	110:   
		   IF Ref_MachineStateModel.Sts_Stopping AND Ref_Unit.EM_Stopping_Done[7] THEN
			  Belt7Seq(Execute:= TRUE, Next:= Seq_Stopping);     
		   ELSE IF NOT (ref_bTransferPut OR HMI_Unit02Simulation) 
                   AND NOT glb_Un02Box.Box[HMI_PrintNo].PrintRequest THEN
				    Belt7Seq(Execute:= TRUE, Next:= 120); 
         		    ELSE IF  NOT glb_Un02Box.Box[HMI_PrintNo].PrintRequest
						     AND NOT glb_Un02Box.Box[0].Valid
							 AND glb_bUnit01BoxNotReady
                             AND NOT glb_bUnit02BoxEmpty THEN
							 Belt7Seq(Execute:= TRUE, Next:= 200); 
					END_IF
				END_IF 
		   END_IF  
  
	120: 
        Ref_Belt.i.Pos:=-150*lrPosCnt; 
		Ref_Belt.i.MoveAbs:=TRUE;		
		Belt7Seq(Execute:= TRUE,Hold:=FALSE, Next:= 130);  
		
	130: 
        IF 	Ref_Belt.o.CmdDone THEN
			lrPosCnt:=lrPosCnt+1;
			Ref_Belt.i.MoveAbs:=FALSE;
			Belt7Seq(Execute:= TRUE,Hold:=FALSE, Next:= 140);  		
		END_IF
		
	140: 
	     IF glb_Un02Box.Box[0].Valid THEN 
			ref_diPrint.0:=TRUE;
		 END_IF

	     FOR iBox:= 63 TO 1 BY -1 DO
			 glb_Un02Box.Box[iBox]:=glb_Un02Box.Box[iBox-1];
		 END_FOR		
		 
		 Belt7Seq(Execute:= TRUE, Hold:=FALSE, Next:= 150);  
		 
	150:	 
		 glb_Un02Box.Box[0].PrintData:='';
		 glb_Un02Box.Box[0].amount:=100;
		 glb_Un02Box.Box[0].Valid:=FALSE;
		 glb_Un02Box.Box[0].PrintRequest:=FALSE;
		 
		 ref_bTransferPut:=TRUE;
		 ref_diPrint:=SHL(ref_diPrint,1);		
		 
		 Belt7Seq(Execute:= TRUE, Hold:=FALSE, Next:= 110);  	
			 
			 
	200:	 
        Ref_Belt.i.Pos:=-150*lrPosCnt; 
		Ref_Belt.i.MoveAbs:=TRUE;		
		Belt7Seq(Execute:= TRUE,Hold:=FALSE, Next:= 210);  		 
		
	210:	 
        IF 	Ref_Belt.o.CmdDone THEN
			lrPosCnt:=lrPosCnt+1;
			Ref_Belt.i.MoveAbs:=FALSE;
			Belt7Seq(Execute:= TRUE,Hold:=FALSE, Next:= 220);  		
		END_IF		 
		 
	220:		 
	     FOR iBox:= 63 TO 1 BY -1 DO
			 glb_Un02Box.Box[iBox]:=glb_Un02Box.Box[iBox-1];
		 END_FOR			
		 ref_diPrint:=SHL(ref_diPrint,1);		
		 Belt7Seq(Execute:= TRUE, Hold:=FALSE, Next:= 110);  

	 
		 
	Seq_stopping: 
	    IF NOT Ref_Belt.o.StandStill THEN
		   Ref_Belt.i.Stop:=TRUE;
		ELSE
		   Belt7Seq(Execute:= TRUE, Next:= 901);  
		END_IF
    901:

       tonBeltSeq(IN:= TRUE, PT:= T#1S, Q=> , ET=> );
	   IF tonBeltSeq.Q THEN
		  tonBeltSeq(IN:= FALSE, PT:= T#1S, Q=> , ET=> );
		  Belt7Seq(Execute:= TRUE, Next:= Seq_StoppingDone);  
	   END_IF
	   
 
	Seq_stoppingDone:	 
	     Ref_Belt.i.disable:=TRUE;
		 IF NOT Ref_MachineStateModel.Sts_Stopping THEN
			Belt7Seq(Execute:= TRUE, Next:= 0);
		 END_IF		 		 
END_CASE
Belt7Seq.Hold := Ref_MachineStateModel.Sts_Held;
END_ACTION

ACTION MainRoution:
EM_No:=8;
IF Ref_Unit.EM_Selected[EM_No] THEN
	IF Ref_MachineStateModel.Sts_Holding THEN
		Ref_Unit.EM_Holding_Done[EM_No]:=TRUE;
		ELSE
		Ref_Unit.EM_Holding_Done[EM_No]:=FALSE;
	END_IF
	IF Ref_MachineStateModel.Sts_UnHolding THEN
		Ref_Unit.EM_UnHolding_Done[EM_No]:=TRUE;
		ELSE
		Ref_Unit.EM_UnHolding_Done[EM_No]:=FALSE;
	END_IF
	
	IF Ref_MachineStateModel.Sts_Suspending THEN
		Ref_Unit.EM_Suspending_Done[EM_No]:=TRUE;
		ELSE
		Ref_Unit.EM_Suspending_Done[EM_No]:=FALSE;
	END_IF
	
	IF Ref_MachineStateModel.Sts_UnSuspending THEN
		Ref_Unit.EM_UnSuspending_Done[EM_No]:=TRUE;
		ELSE
		Ref_Unit.EM_UnSuspending_Done[EM_No]:=FALSE;
	END_IF

	IF Ref_MachineStateModel.Sts_Resetting AND Belt7Seq.Now=100 THEN
       Ref_Unit.EM_Resetting_Done[EM_No]:=TRUE;   
       ELSE   
       Ref_Unit.EM_Resetting_Done[EM_No]:=FALSE;   
	END_IF
	
	IF Ref_MachineStateModel.Sts_Clearing THEN
		Ref_Unit.EM_Clearing_Done[EM_No]:=TRUE;
		ELSE
		Ref_Unit.EM_Clearing_Done[EM_No]:=FALSE;  
	END_IF
		
	IF Ref_MachineStateModel.Sts_Starting THEN
	   Ref_Unit.EM_Starting_Done[EM_No]:=TRUE;
	   ELSE
	   Ref_Unit.EM_Starting_Done[EM_No]:=FALSE;
	END_IF
		
	IF Ref_MachineStateModel.Sts_Stopping AND Belt7Seq.Now=1000 THEN
       Ref_Unit.EM_Stopping_Done[EM_No]:=TRUE;
	   ELSE
	   Ref_Unit.EM_Stopping_Done[EM_No]:=FALSE;
	END_IF
	
	IF Ref_MachineStateModel.Sts_Aborting THEN	
		Belt7Seq(Execute:= TRUE, Next:= 0);
        IF  NOT Ref_Belt.o.StandStill THEN
			Ref_Belt.i.Stop :=TRUE;
			ELSE 
			Ref_Belt.i.Stop :=FALSE;
		END_IF
		
		IF  tonAbortingWatchDog.Q THEN 
			Ref_Unit.EM_Aborting_Done[EM_No]:=TRUE;
			Ref_Belt.i.Disable:=TRUE;
		END_IF
	END_IF
	tonAbortingWatchDog(IN:= Ref_MachineStateModel.Sts_Aborting, PT:=T#3S , Q=> , ET=> );	
//////////////////////////////////////////////////////////////////////////////////////////////
	CM02_Belt();
ELSE
	 Belt7Seq(Execute:= TRUE, Next:= 0);
END_IF
END_ACTION

ACTION SR999_FaultHandler:
;
END_ACTION

END_PROGRAM

// ---- POUs/Debug/DebugPro.TcPOU
PROGRAM DebugPro
VAR
    MC_MoveAbsolute_Axis: ARRAY[1..8] OF MC_MoveAbsolute ;
	MC_MoveAdditive_Axis: ARRAY[1..8] OF MC_MoveAdditive;
	MC_MoveRelative_Axis: array[1..8] of MC_MoveRelative;
	iDebug: INT;
	iDebugCyc: INT;
	tonDebug: Ton;
END_VAR

MC_MoveAbsolute_Axis[1](
	Axis:= arRealAxisAdmin[47].Axis, 
	Execute:= , 
	Position:= , 
	Velocity:= 10, 
	Acceleration:= 10, 
	Deceleration:= 10, 
	Jerk:= 10000, 
	BufferMode:= , 
	Options:= , 
	Done=> , 
	Busy=> , 
	Active=> , 
	CommandAborted=> , 
	Error=> , 
	ErrorID=> );

MC_MoveAbsolute_Axis[2](
	Axis:= arRealAxisAdmin[47].Axis, 
	Execute:= , 
	Position:= , 
	Velocity:= 100, 
	Acceleration:= 1000, 
	Deceleration:= 1000, 
	Jerk:= 10000, 
	BufferMode:= , 
	Options:= , 
	Done=> , 
	Busy=> , 
	Active=> , 
	CommandAborted=> , 
	Error=> , 
	ErrorID=> );	
	
MC_MoveAdditive_Axis[1](
	Axis:= arRealAxisAdmin[47].Axis, 
	Execute:= , 
	Distance:= , 
	Velocity:= 10, 
	Acceleration:= 100, 
	Deceleration:= 100, 
	Jerk:= 10000, 
	BufferMode:= , 
	Options:= , 
	Done=> , 
	Busy=> , 
	Active=> , 
	CommandAborted=> , 
	Error=> , 
	ErrorID=> );

MC_MoveAdditive_Axis[2](
	Axis:= arRealAxisAdmin[47].Axis, 
	Execute:= , 
	Distance:= , 
	Velocity:= 10, 
	Acceleration:= 100, 
	Deceleration:= 100, 
	Jerk:= 10000, 
	BufferMode:= , 
	Options:= , 
	Done=> , 
	Busy=> , 
	Active=> , 
	CommandAborted=> , 
	Error=> , 
	ErrorID=> );
		
MC_MoveRelative_Axis[1](
	Axis:= arRealAxisAdmin[47].Axis, 
	Execute:= , 
	Distance:= , 
	Velocity:= 10, 
	Acceleration:= 100, 
	Deceleration:= 100, 
	Jerk:= 10000, 
	BufferMode:= , 
	Options:= , 
	Done=> , 
	Busy=> , 
	Active=> , 
	CommandAborted=> , 
	Error=> , 
	ErrorID=> );	
	
MC_MoveRelative_Axis[2](
	Axis:= arRealAxisAdmin[47].Axis, 
	Execute:= , 
	Distance:= , 
	Velocity:= 10, 
	Acceleration:= 100, 
	Deceleration:= 100, 
	Jerk:= 10000, 
	BufferMode:= , 
	Options:= , 
	Done=> , 
	Busy=> , 
	Active=> , 
	CommandAborted=> , 
	Error=> , 
	ErrorID=> );	
	
CASE iDebug OF
	
10: MC_MoveAbsolute_Axis[1].Position:=100;
    MC_MoveAbsolute_Axis[1].Execute:=TRUE;
	IF MC_MoveAbsolute_Axis[1].Active THEN
	   MC_MoveAbsolute_Axis[1].Execute:=FALSE;
       iDebug:=20;
	END_IF
20:
    MC_MoveAbsolute_Axis[2].Position:=200;
    MC_MoveAbsolute_Axis[2].Execute:=TRUE;
	IF MC_MoveAbsolute_Axis[2].Active THEN
	   MC_MoveAbsolute_Axis[2].Execute:=FALSE;
	   iDebug:=iDebugCyc;
	END_IF
		
100: MC_MoveAdditive_Axis[1].Distance:=100;
    MC_MoveAdditive_Axis[1].Execute:=TRUE;
	IF MC_MoveAdditive_Axis[1].Active THEN
	   MC_MoveAdditive_Axis[1].Execute:=FALSE;
       iDebug:=200;
	END_IF
200:
    MC_MoveAdditive_Axis[2].Distance:=100;
    MC_MoveAdditive_Axis[2].Execute:=TRUE;
	IF MC_MoveAdditive_Axis[2].Active THEN
	   MC_MoveAdditive_Axis[2].Execute:=FALSE;
	   iDebug:=iDebugCyc;
	END_IF	
	
	
1000: MC_MoveRelative_Axis[1].Distance:=100;
    MC_MoveRelative_Axis[1].Execute:=TRUE;
	IF MC_MoveRelative_Axis[1].Active THEN
	   MC_MoveRelative_Axis[1].Execute:=FALSE;
       iDebug:=1100;
	END_IF
	
1100: 
     tonDebug(IN:= TRUE, PT:= T#1S, Q=> , ET=> );
	 IF tonDebug.Q THEN
		 tonDebug(IN:= FALSE, PT:= T#1S, Q=> , ET=> ); 
		 iDebug:=2000;
	 END_IF

	
2000:
    MC_MoveRelative_Axis[2].Distance:=100;
    MC_MoveRelative_Axis[2].Execute:=TRUE;
	IF MC_MoveRelative_Axis[2].Active THEN
	   MC_MoveRelative_Axis[2].Execute:=FALSE;
	   iDebug:=iDebugCyc;
	END_IF		
END_CASE

END_PROGRAM

// ---- Add-On-Instructions/AOI_CountersAdmin.TcPOU
FUNCTION_BLOCK AOI_CountersAdmin
VAR_INPUT
	Enable: BOOL; //启用
	Execute: BOOL; //数粒信号
	Reset: bool; //重置
    In_Total: DINT; //计划生产总数
	Quantity: DINT;
	Clear: BOOL;//清除故障
	SkipAlarm: BOOL;
	CheckTime: DINT;
    CheckCnt: BOOL;
	ManualCnt: BOOL;
END_VAR
VAR_OUTPUT
	DropVibrator_Wrk: BOOL;//落料启动
	CircleVibrator_Wrk: BOOL;//圆震启动
	LineVibrator_Wrk: BOOL;//直震启动
	Warning: BOOL;	
	Busy: BOOL;//数粒中
	Error: BOOL; //报警
	ErrorID: DINT;//报警代码;	
	InitDone: BOOL;//初始化完成
	Out_Total: DINT;//实际生产数量
	Complete: BOOL; //生产完成
	CntUp: DINT;
	ProcessTime : DINT;//
	Speed: REAL;
END_VAR
VAR
	iAxisAct: INT;	
	tonHighCheck: TON;
	tonLowCheck: TON;
	tonLackCheck: TON;
	tonWatchDog: TON;
	tonProcess: TON;
	tonEnable: TON;
	rt_Exe: R_TRIG;	
	aoi_DropSensor: AOI_Sensoradmin;
	aoi_LowSensor: AOI_Sensoradmin;
	aoi_HighSensor: AOI_Sensoradmin;	
	lrPosAdd: LREAL;
	rt_Clear: R_TRIG; 
	rt_Drop: R_TRIG;
	rtLowCheck: R_trig;
	toncheck: TON;
	diLastTargetCnt: DINT;
	QuantityBuffer: DINT;
	tonDropDelay: Ton;
	diCheckFaultCnt: DINT;
	diFaultCnt: ARRAY[0..64] OF dint;
	i: INT;
END_VAR
VAR_IN_OUT
	Axis: UDT_AxisAdmin;//数粒伺服
	DropSensor: UDT_SensorAdmin;//缺料检测
	LowSensor: UDT_SensorAdmin;//低料位检测
	HighSensor: UDT_SensorAdmin;//高料位检测
	Cylinder: UDT_CylinderAdmin;//
	DropFlag: BOOL;//
END_VAR

rt_Exe(CLK:=Execute , Q=> );
rt_Drop(CLK:= DropSensor.o.Value, Q=> );
tonEnable(IN:= Enable, PT:= T#3S, Q=> , ET=> );
IF NOT Enable THEN		
	DropVibrator_Wrk:=FALSE;//震动盘启动
	CircleVibrator_Wrk:=FALSE;
	LineVibrator_Wrk:=FALSE;	
END_IF

IF Enable THEN
   IF NOT HighSensor.o.Value  AND NOT Complete THEN
	  DropVibrator_Wrk:=TRUE;//落料震动盘启动
	  ELSE
	  DropVibrator_Wrk:=FALSE;//
   END_IF
   IF NOT LowSensor.o.Value AND NOT Complete  THEN	  
	   CircleVibrator_Wrk:=TRUE;//圆震动盘启动
	   ELSE
	   CircleVibrator_Wrk:=FALSE;	   
   END_IF	
   CircleVibrator_Wrk:= TRUE;
   LineVibrator_Wrk:= TRUE;//直震动盘启动常开
ELSE
   DropVibrator_Wrk:=FALSE;
   LineVibrator_Wrk:= FALSE;
   CircleVibrator_Wrk:= FALSE;
END_IF

IF reset THEN
	Complete:=FALSE;
	Out_Total:=0;
END_IF

rt_Clear(CLK:= Clear, Q=> );
IF rt_Clear.Q THEN
   Error:=FALSE;
END_IF

IF Enable AND Quantity=0 THEN
	IF DropFlag THEN
	   DropFlag:=FALSE;
	END_IF
END_IF

CASE iAxisAct OF
	0: 
        Busy:=FALSE;
		IF Out_Total<In_Total AND Quantity<>0 AND tonEnable.Q THEN
		   QuantityBuffer:=Quantity;
		   iAxisAct:=10;
		ELSE IF Out_Total=In_Total THEN
				Complete:=TRUE;
		     END_IF
		END_IF

	10:
	    IF QuantityBuffer>20 THEN
		   QuantityBuffer:=QuantityBuffer-20;
		   iAxisAct:=11;
		ELSE
           iAxisAct:=12;   
	    END_IF
	   
	11:
	    Busy:=TRUE;
		CntUp:=0;
	    lrPosAdd:=20*360/24; 
		diLastTargetCnt:=20;
	    Axis.i.Pos:=lrPosAdd;
		iAxisAct:=20;
		
	12: 
	    Busy:=TRUE;
		CntUp:=0;
	    lrPosAdd:=QuantityBuffer*360/24; 
		diLastTargetCnt:=QuantityBuffer;
		QuantityBuffer:=0;
	    Axis.i.Pos:=lrPosAdd;
		iAxisAct:=20;
	    
	20:
	    Axis.i.MoveAdd:=TRUE;
	    tonProcess(IN:=TRUE , PT:=T#100S , Q=> , ET=> );
	    ProcessTime:= TIME_TO_DINT(tonProcess.ET);
		IF Axis.o.CmdDone OR Axis.o.Error THEN
		   Axis.i.MoveAdd:=FALSE;
		   iAxisAct:=30;
		   tonProcess(IN:=FALSE , PT:=T#100S , Q=> , ET=> );
		   Speed:=1000/DINT_TO_REAL(ProcessTime);
		END_IF
	30:
		toncheck(IN:= TRUE, PT:= DINT_TO_TIME(CheckTime), Q=> , ET=> );
		
	    IF NOT SkipAlarm AND toncheck.Q AND CntUp<1  THEN
		   Error:=TRUE;
		END_IF
		IF NOT CheckCnt AND toncheck.Q AND CntUp <> diLastTargetCnt THEN
		   Error:=TRUE;
		END_IF
		
		IF toncheck.Q AND CntUp <> diLastTargetCnt THEN
		   diCheckFaultCnt:=diCheckFaultCnt+1;
		   diFaultCnt[i]:=CntUp;
		   i:=i+1;
		   IF i>60 THEN
			   i:=0;
		   END_IF
		END_IF
		
		
		IF (SkipAlarm AND CheckCnt)OR toncheck.Q THEN
		   toncheck(IN:= FALSE, PT:= DINT_TO_TIME(CheckTime), Q=> , ET=> );
           iAxisAct:=100;
		END_IF
		
	100:	
	    Busy:=FALSE;
		IF NOT Cylinder.i.OutSensor AND NOT Cylinder.i.InSensor THEN
		   Cylinder.i.ActiveIn:=TRUE;
		   Cylinder.i.ActiveOut:=FALSE;
		END_IF
		
		IF DropFlag AND NOT Error THEN
		   IF Cylinder.i.OutSensor THEN
		      iAxisAct:=110;
           END_IF	
		   IF Cylinder.i.InSensor THEN
		      iAxisAct:=120;
           END_IF	
		END_IF		
		IF Error AND rt_Drop.Q THEN
		   iAxisAct:=101;
		END_IF
		
		IF Reset THEN
		   iAxisAct:=0;
        END_IF
		
	101:	
		Axis.i.Pos:=360/24;
	    Axis.i.MoveAdd:=TRUE;
		IF Axis.o.CmdDone OR Axis.o.Error THEN
		   Axis.i.MoveAdd:=FALSE;
		   iAxisAct:=102;
		END_IF		
	102:
	    tonDropDelay(IN:= TRUE, PT:= T#1S, Q=> , ET=> );
		IF tonDropDelay.Q THEN
			tonDropDelay(IN:= FALSE, PT:= T#1S, Q=> , ET=> );
			iAxisAct:=100;
		END_IF
		
	110: 
	    Cylinder.i.ActiveIn:=TRUE;
		Cylinder.i.ActiveOut:=FALSE;
		IF Cylinder.i.InSensor THEN
			iAxisAct:=200;
		END_IF
		
	120:
	    Cylinder.i.ActiveIn:=FALSE;
		Cylinder.i.ActiveOut:=TRUE;
		IF Cylinder.i.OutSensor THEN
			iAxisAct:=200;
		END_IF	
	200:
	    IF QuantityBuffer=0 THEN
		   iAxisAct:=300;
		ELSE 
		   iAxisAct:=10;
		END_IF
	
	300:
	    Out_Total:=Out_Total+1; 
        DropFlag:=FALSE;
	    iAxisAct:=0;
	
END_CASE

tonHighCheck(IN:= NOT HighSensor.o.Value AND Enable AND Quantity<>0 , PT:=T#15S , Q=> , ET=> );
tonLowCheck(IN:= NOT LowSensor.o.Value  AND Enable, PT:=T#5S , Q=> , ET=> );
rtLowCheck(CLK:= LowSensor.o.Value, Q=> );

IF rtLowCheck.Q THEN
   CntUp:=CntUp+1;
END_IF

Warning:= tonHighCheck.Q AND NOT Error ;

aoi_DropSensor(Admin:= DropSensor);
aoi_HighSensor(Admin:= HighSensor);
aoi_LowSensor(Admin:= LowSensor);

END_FUNCTION_BLOCK

// ---- Add-On-Instructions/AOI_DI.TcPOU
FUNCTION_BLOCK AOI_DI
VAR_INPUT
	ON: BOOL;
	OFF: BOOL;
	NAME: STRING := 'Not use';
	LINK: BOOL;
END_VAR
VAR_OUTPUT
	VALUE: BOOL;
	R_TRIG: BOOL;
	F_TRIG: BOOL;
END_VAR
VAR
	rtON: R_TRIG;
	rtOFF: R_TRIG;
	ftON: F_TRIG;
	ftOFF: F_TRIG;	
	rtValue: R_TRIG;
	ftValue: F_TRIG;

END_VAR

VALUE:= (ON OR LINK) AND NOT OFF; 
rtValue(CLK:=VALUE);
ftValue(CLK:=VALUE);
R_TRIG:=rtValue.Q;
F_TRIG:=ftValue.Q; 
rtON(CLK:=ON);
(*
IF rtON.Q THEN
	OFF:=FALSE;
	ON:=TRUE;	
END_IF
rtOFF(CLK:=OFF);
IF rtOFF.Q THEN
	ON:=FALSE;
	OFF:=TRUE;
END_IF

rtOFF(CLK:= OFF, Q=> );

IF ftOFF.Q THEN
	OFF:=FALSE;
END_IF

rtON(CLK:= ON, Q=> );

IF ftON.Q THEN
	ON:=FALSE;
END_IF

*)
IF ON AND OFF THEN
	ON:=FALSE;
	OFF:=FALSE;	
END_IF

END_FUNCTION_BLOCK

// ---- Add-On-Instructions/AOI_DO.TcPOU
FUNCTION_BLOCK AOI_DO
VAR_INPUT
	ON: BOOL;
	OFF: BOOL;
	NAME: STRING := 'Not use';
	VALUE: BOOL;
END_VAR
VAR_OUTPUT
	LINK: BOOL;
	R_TRIG: BOOL;
	F_TRIG: BOOL;
END_VAR
VAR
	rtON: R_TRIG;
	rtOFF: R_TRIG;
	rtValue: R_TRIG;
	ftValue: F_TRIG;
END_VAR

LINK:=  (ON OR  VALUE)   AND NOT OFF; 

rtValue(CLK:=VALUE);
ftValue(CLK:=VALUE);
R_TRIG:=rtValue.Q;
F_TRIG:=ftValue.Q;
rtON(CLK:=ON);
(*
IF rtON.Q THEN
	OFF:=FALSE;
	On:=TRUE;
END_IF
rtOFF(CLK:=OFF);
IF rtOFF.Q THEN
	ON:=FALSE;
	OFF:=TRUE;
END_IF
*)
IF on AND off THEN
	ON:=FALSE;
	OFF:=FALSE;	
END_IF

END_FUNCTION_BLOCK

// ---- Add-On-Instructions/AOI_DeltaScaraRobot.TcPOU
FUNCTION_BLOCK AOI_DeltaScaraRobot
VAR_INPUT
END_VAR
VAR_OUTPUT
END_VAR
VAR
	rtStart: R_trig;
	rtStop: R_Trig;
	rtHold: R_Trig;
END_VAR
VAR_IN_OUT
	Scara: UDT_Scara;
END_VAR

IF Scara.i.Auto THEN
   Scara.Di_[1][4]:=0;
   Scara.Di_[1][5]:=1;   
   ELSE IF Scara.i.T2  THEN
	      Scara.Di_[1][4]:=1;
          Scara.Di_[1][5]:=1;     
         END_IF 		
END_IF

IF rtStart.Q  THEN
   Scara.Di_[1][6]:=1;
   Scara.Di_[1][7]:=1;
END_IF   
IF Scara.i.Stop THEN
   Scara.Di_[1][6]:=1;
   Scara.Di_[1][7]:=0;
END_IF   
IF rtHold.Q THEN
	Scara.Di_[1][6]:=0;
	Scara.Di_[1][7]:=1;
END_IF


rtStart(CLK:=Scara.i.Start , Q=> );
rtStop(CLK:=Scara.i.Stop , Q=> );
rtHold(CLK:=Scara.i.Hold , Q=> );

Scara.Di_[1][1]:=NOT Scara.i.Estop AND NOT Scara.i.Shutdown ;
Scara.Di_[1][2]:=NOT Scara.i.Estop;
Scara.Di_[1][3]:=Scara.i.Reset;
Scara.Di_[1][8]:=Scara.i.reset OR scara.i.FuctionReset;

Scara.o.Error:=Scara.Do_[1][1];
Scara.o.Enable:=Scara.Do_[1][2];
Scara.o.InPos:=Scara.Do_[1][3];
Scara.o.FuctionHold:=Scara.Do_[1][4];
Scara.o.ProRunning:=Scara.Do_[1][5] AND Scara.Do_[1][6];
Scara.o.Held:=NOT Scara.Do_[1][5] AND Scara.Do_[1][6];
Scara.o.ProStopped:= Scara.Do_[1][5] AND NOT Scara.Do_[1][6];

Scara.Di_[2][1]:=Scara.i.ProFaultClear;
Scara.Di_[2][2]:=Scara.i.ProPick;
Scara.Di_[2][3]:=Scara.i.ProDepart;
Scara.Di_[2][4]:=Scara.i.ProPut;
Scara.Di_[2][5]:=Scara.i.LoopStop;//循环停止

Scara.o.ProFault:=Scara.Do_[2][1];
Scara.o.ProPickDone:=Scara.Do_[2][2];
Scara.o.ProPutDone:=Scara.Do_[2][3];
Scara.o.ProDepartDone:=Scara.Do_[2][4];
Scara.o.LoopStopDone:=Scara.Do_[2][5];//循环完成
Scara.o.ResettingDone:=Scara.Do_[2][6];//复位完成

END_FUNCTION_BLOCK

// ---- Add-On-Instructions/AOI_Heat.TcPOU
FUNCTION_BLOCK AOI_Heat
VAR_INPUT
	Enable: BOOL;
	PV: REAL;
	SV: REAL;
	Pi: REAL:=0.5;
	Kp: REAL:= 0.3;
	Ki: REAL:= 0.6;
	Kd: REAL:=0.5;
	Reset: BOOL;
	HighLimit: REAL;
	LowLimit: REAL;
	MaxHeatTime: DINT;	
END_VAR
VAR_OUTPUT
	Active: BOOL;
	Actuator: BOOL;
	Error: BOOL;
	ErrorID: DINT;
END_VAR
VAR
	tonAct: TON;
	tonHeatError: TON;
	rtActive: R_Trig;
	PV_Old: REAL;
	CV: REAL;
	tonHeatting: TON;
	iAct: INT;
	bErrorCheck: BOOL;
	rDiff: REAL;
	tonReset: Ton;
	xReset: BOOL;
	rDiffOld: REAL;
	blinkHeat: BLINK;

	diHeatTime: DINT;
	Ut: REAL;

	iPID: INT;
	rErrSum: REAL;
	rErr: REAL;
	rOldErr: REAL;
	tonPID: TON;
	tonActive: TON;	
	iCyc: INT;

	iKdCount: INT;
	Ui: REAL;
	tonHighAlarm: Ton;
	tonLowAlarm: Ton;	
END_VAR

CASE iAct OF
	0:
       IF Enable THEN
		  iAct:=10;
	   END_IF
	   Active:=FALSE;
	10:
       IF NOT ErrorID.0 THEN
			IF SV>PV THEN
			   Active:=TRUE;
			   PV_Old:=PV;
			   //rDiffOld:=rDiff;
			   //rDiff:=SV-PV;
			   //CV:=(SV-PV)*1000*Pi;
			   iAct:=20;
			END_IF
        ELSE 
 	        Active:=FALSE;
		END_IF	
		IF NOT Enable THEN
		   iAct:=0;
		END_IF  
    20: 
	(*
	    tonAct(IN:=TRUE , PT:=REAL_TO_TIME(CV), Q=> , ET=> );
		IF tonAct.Q OR PV>= SV THEN
		   tonAct(IN:=FALSE , PT:= REAL_TO_TIME(CV), Q=> , ET=> );	
		   Active:=FALSE;
		   IF PV <PV_OLD THEN
	          bErrorCheck:=TRUE;
			  ELSE
		      bErrorCheck:=FALSE;
           END_IF
		   iAct:=30;
		END_IF
	 *)
		IF PV>= SV+1 THEN
			Active:=FALSE;
			iAct:=10;
		END_IF
		IF PV <PV_OLD THEN
			  bErrorCheck:=TRUE;
			  ELSE
			  bErrorCheck:=FALSE;
		END_IF
    30:
		IF (PV-PV_OLD) < rDiff/2 THEN
			iAct:=10;
		ELSE
			iAct:=40;
		END_IF
	40:	
		tonAct(IN:=TRUE , PT:= REAL_TO_TIME(CV/5), Q=> , ET=> );
		IF tonAct.Q THEN
		tonAct(IN:=FALSE , PT:= REAL_TO_TIME(CV/5), Q=> , ET=> );
			iAct:=10;
		END_IF
END_CASE
(*
tonHeatError(IN:= bErrorCheck, PT:=T#10M, Q=> , ET=> );
IF tonHeatError.Q  THEN
   bErrorCheck:=FALSE;
   Error:=TRUE;
   ErrorID.2:=1;
END_IF
*)
tonHighAlarm(IN:= (PV > (SV+HighLimit) OR PV > 300), PT:=T#1S , Q=> , ET=> );
tonLowAlarm(IN:= (PV <(SV-LowLimit)), PT:=T#1S , Q=> , ET=> );
IF NOT xReset THEN
	IF tonHighAlarm.Q THEN
	   Error:=TRUE;
	   ErrorID.0:=1;
	END_IF
	
	IF tonLowAlarm.Q  THEN
		Error:=TRUE;
		ErrorID.1:=1;
	END_IF
END_IF	

diHeatTime:=REAL_TO_DINT(CV)/100*MaxHeatTime;

blinkHeat(TimeH:= , TimeL:= , OUT=> );



IF Reset OR NOT Enable THEN
	xReset:=TRUE;
	Error:=FALSE; 
	ErrorID:=0;
END_IF

tonReset(IN:= xReset, PT:= T#1S, Q=> , ET=> );
IF tonReset.q THEN
   xReset:=FALSE;
END_IF

(*
CASE iPID OF 
	0: 
       rOldErr:=rErr;
       rErr:=SV-PV;
	   rErrSum:=rErrSum+rErr;
	   iKdCount:=iKdCount+1;       
	   IF iKdCount>Ki THEN
          Ui:=rErrSum;	
		  iKdCount:=0;
          rErrSum:=0;  
	   END_IF
	   Ut:=Kp*rErr+Ui+Kd*(rErr-rOldErr);
	 
	   IF Ut>100 THEN
		   Ut:=100;
	   ELSE IF Ut<0 THEN
		       Ut:=0;
		    END_IF
	   END_IF
	   iPID:=100;
	   
    100: 
	   IF TIME_TO_REAL(tonActive.ET) < Ut/100*1000 AND NOT ErrorID.0 THEN
		   Actuator:=TRUE;
		   ELSE
		   Actuator:=FALSE;   
	   END_IF
	
       tonActive(IN:= TRUE, PT:= T#1S, Q=> , ET=> );
	   IF tonActive.Q THEN
		  tonActive(IN:= FALSE, PT:= T#1S, Q=> , ET=> );  
		  iPID:=0;
	   END_IF	
END_CASE
*)

END_FUNCTION_BLOCK

// ---- Add-On-Instructions/ethercatinfo_read.TcPOU
FUNCTION_BLOCK ethercatinfo_read
VAR_INPUT
	netID AT %I*:Tc2_System.T_AmsNetIdArr;							//硬件网络的AMSnetID
	nEcMasterDeviceId AT %I*:UINT;											//主站的deviceID
END_VAR
VAR_OUTPUT
	slaveAddresses    : ARRAY[0..255] OF UINT;						//读取的从站地址（以数组保存）
	devStates           : ARRAY[0..255] OF ST_EcSlaveState;		//读取的从站状态机
	slavenames			: ARRAY[0..255] OF T_MaxString;			//读取从站名字
    color					: ARRAY[0..255] OF DWORD;					//显示图标的颜色
	nSlaves           : UINT := 0;														//从站个数
END_VAR
VAR
	i:INT;
	i1:INT;
	NAN:Tc2_System.T_MaxString;											//复位变量
	ton1:Tc2_Standard.TON;														//读取时钟触发器
	bExecute          :  BOOL;															//触发位
	fb_getalladdr:Tc2_EtherCAT.FB_EcGetAllSlaveAddr;		//读取从站地址的功能块 https://infosys.beckhoff.com/content/1033/tcplclib_tc2_ethercat/9007199311752331.html?id=8671424095593379685
	fb_getallstate:Tc2_EtherCAT.FB_EcGetAllSlaveStates;		//读取从站状态机的功能块 https://infosys.beckhoff.com/content/1033/tcplclib_tc2_ethercat/9007199311770635.html?id=2217456128990928132
	fb_getallname: IOF_GetBoxNameByAddr;							//读取从站名称 https://infosys.beckhoff.com/content/1033/tcplclib_tc2_iofunctions/9007199313832971.html?id=4102389766817989774
END_VAR

ton1(IN:= NOT ton1.Q, PT:= T#0.5S, Q=> bExecute, ET=> );

fb_getalladdr(//读取从站地址
	sNetId:= F_CreateAmsNetId(netID), //网络netID
	pAddrBuf:= ADR(slaveAddresses), //寄存器地址
	cbBufLen:= SIZEOF(slaveAddresses), 
	bExecute:= bExecute, 
	nSlaves=> nSlaves);//从站个数
	
fb_getallstate(//读取从站状态机
	sNetId:= F_CreateAmsNetId(netID), //网络地址
	pStateBuf:= ADR(devStates), //寄存器地址
	cbBufLen:= SIZEOF(devStates), 
	bExecute:= bExecute, 
	nSlaves=> );

fb_getallname(//读取从站名称
	NETID:= , 
	DEVICEID:=nEcMasterDeviceId, //device number
	BOXADDR:=  slaveAddresses[i], //从站号
	BOXNAME=> slavenames[i]);//返回从站名

IF slaveAddresses[i]>0 AND NOT fb_getallname .start THEN//反复触发功能块
	fb_getallname.START:=TRUE;
ELSIF slaveAddresses[i+1]>0 AND NOT fb_getallname.BUSY THEN
		i:=i+1;
		fb_getallname.START:=FALSE;
END_IF

FOR i1:=0 TO  nSlaves BY 1 DO//颜色变量触发逻辑
CASE devStates [i1].deviceState OF
	1: color[i1]:=16#FFFF0000;
	2: color[i1]:=16#FFFFFF00;
	4: color[i1]:=16#FF88FF00;
	8: color[i1]:=16#FF00FF00;
	ELSE
	color[i1]:=16#FFFFFFFF;
END_CASE
END_FOR

END_FUNCTION_BLOCK

// ---- Add-On-Instructions/systeminfo_MDP_read.TcPOU
FUNCTION_BLOCK systeminfo_MDP_read
VAR_INPUT
	excute:BOOL;
	moduletype:WORD;  //module类型，参考https://infosys.beckhoff.com/content/1033/devicemanager/99079192065133835.html?id=1049129283645184856
	tableID:BYTE;//附表标号
	sbidxcount:USINT:=20;
	startidx:INT;
	outputadr:PVOID;
	outputsiz:UDINT;
END_VAR
VAR_OUTPUT
	bbusy:BOOL;
	berror:BOOL;
	nerrID1:UDINT;
	nerrID2:UDINT;
END_VAR
VAR
	excute1,excute2:BOOL;													//触发位
	dsbuf:ARRAY[0..254] OF BYTE;										//	寄存器数组
	trig:Tc2_Standard.F_TRIG;
	MDPaddr:Tc2_MDP.ST_MDP_Addr;								//功能块
	FB_scanmodule:Tc2_MDP.FB_MDP_ScanModules;	//https://infosys.beckhoff.com/content/1033/tcplclib_tc2_mdp/27021597942949259.html?id=8338783758843393121
	FB_read:Tc2_MDP.FB_MDP_ReadModuleContent;	//https://infosys.beckhoff.com/content/1033/tcplclib_tc2_mdp/27021597942946187.html?id=6623212347933124917
END_VAR

excute1:=excute;
trig(CLK:= FB_scanmodule.bBusy, Q=>excute2 );
bbusy :=FB_scanmodule.bBusy AND FB_read.bBusy;
berror :=FB_scanmodule .bError AND FB_read.bError;

FB_scanmodule(
	bExecute:= excute1, 
	nModuleType:=moduletype, 
	iModIdx:= 0, 
	tTimeout:= , 
	sAmsNetId:= , 
	bBusy=> , 
	bError=> , 
	nErrID=> nerrID1, 
	nDynModuleId=> , 
	iModuleTypeCount=> , 
	iModuleCount=> );

MDPaddr.nArea:=16#8;
MDPaddr.nModuleId:=FB_scanmodule.nDynModuleId;
MDPaddr.nTableId:=tableID;//附表标号

FB_read(
	bExecute:= excute2, 
	stMDP_DynAddr:= MDPaddr, 
	iSubIdxCount:= sbidxcount, //附表长度
	pDstBuf:= ADR(dsbuf), 
	cbDstBufLen:= SIZEOF(dsbuf), 
	tTimeout:= , 
	sAmsNetId:= , 
	bBusy=> , 
	bError=> , 
	nErrID=> nerrID2, 
	iErrPos=> , 
	arrStartIdx=> );
	
Tc2_System.MEMCPY(outputadr,ADR(dsbuf[FB_read.arrStartIdx[startidx(*附表参数号，即subindex*)]]),outputsiz);//将对应的参数赋值给相应的变量

END_FUNCTION_BLOCK

// ---- POUs/POUCheck/CheckBounds.TcPOU
// 隐含生成代码：不要编辑
FUNCTION CheckBounds : DINT
VAR_INPUT
	index, lower, upper: DINT;
END_VAR

// 隐含生成代码：这里只是对代码实现的建议
{noflow}
IF  index < lower THEN
	CheckBounds := lower;
ELSIF  index > upper THEN
	CheckBounds := upper;
ELSE  
	CheckBounds := index;
END_IF
{flow}

END_FUNCTION

// ---- POUs/POUCheck/CheckDivDInt.TcPOU
// 隐含生成代码：不要编辑
FUNCTION CheckDivDInt : DINT
VAR_INPUT
	divisor:DINT;
END_VAR

// 隐含生成代码：这里只是对代码实现的建议
{noflow}
IF divisor = 0 THEN
	CheckDivDInt:=1;
ELSE
	CheckDivDInt:=divisor;
END_IF;
{flow}

END_FUNCTION

// ---- POUs/POUCheck/CheckDivLInt.TcPOU
// 隐含生成代码：不要编辑
FUNCTION CheckDivLInt : LINT
VAR_INPUT
	divisor:LINT;
END_VAR

// 隐含生成代码：这里只是对代码实现的建议
{noflow}
IF divisor = 0 THEN
	CheckDivLInt:=1;
ELSE
	CheckDivLInt:=divisor;
END_IF;
{flow}

END_FUNCTION

// ---- POUs/POUCheck/CheckDivLReal.TcPOU
// 隐含生成代码：不要编辑
FUNCTION CheckDivLReal : LREAL
VAR_INPUT
	divisor:LREAL;
END_VAR

// 隐含生成代码：这里只是对代码实现的建议
{noflow}
IF divisor = 0 THEN
	CheckDivLReal:=1;
ELSE
	CheckDivLReal:=divisor;
END_IF;
{flow}

END_FUNCTION

// ---- POUs/POUCheck/CheckDivReal.TcPOU
// 隐含生成代码：不要编辑
FUNCTION CheckDivReal : REAL
VAR_INPUT
	divisor:REAL;
END_VAR

// 隐含生成代码：这里只是对代码实现的建议
{noflow}
IF divisor = 0 THEN
	CheckDivReal:=1;
ELSE
	CheckDivReal:=divisor;
END_IF;
{flow}

END_FUNCTION

// ---- POUs/POUCheck/CheckLRangeSigned.TcPOU
// 隐含生成代码：不要编辑
FUNCTION CheckLRangeSigned : LINT
VAR_INPUT
	value, lower, upper: LINT;
END_VAR

// 隐含生成代码：这里只是对代码实现的建议
{noflow}
IF (value < lower) THEN
	CheckLRangeSigned := lower;
ELSIF(value > upper) THEN
	CheckLRangeSigned := upper;
ELSE
	CheckLRangeSigned := value;
END_IF

{flow}

END_FUNCTION

// ---- POUs/POUCheck/CheckLRangeUnsigned.TcPOU
// 隐含生成代码：不要编辑
FUNCTION CheckLRangeUnsigned : ULINT
VAR_INPUT
	value, lower, upper: ULINT;
END_VAR

// 隐含生成代码：这里只是对代码实现的建议
{noflow}
IF (value < lower) THEN
	CheckLRangeUnsigned := lower;
ELSIF(value > upper) THEN
	CheckLRangeUnsigned := upper;
ELSE
	CheckLRangeUnsigned := value;
END_IF
{flow}

END_FUNCTION

// ---- POUs/POUCheck/CheckPointer.TcPOU
// 隐含生成代码：不要编辑
FUNCTION CheckPointer : POINTER TO BYTE
VAR_INPUT 
	ptToTest : POINTER TO BYTE; // 指针的目标地址
	iSize : DINT;		        // 指针指向的类型大小。（例如：POINTER TO ARRAY [0..9] OF INT为20）
	iGran : DINT;		        // 指针访问的粒度，即指针指向的类型中最大的非结构数据类型的大小。（例如：POINTER TO ARRAY [0..9] OF INT为2）
	bWrite: BOOL;		        // 指示读或写权限。TRUE=写权限。
END_VAR

// 没有标准的实现方式。在此处输入代码
CheckPointer := ptToTest;
{flow}

END_FUNCTION

// ---- POUs/POUCheck/CheckRangeSigned.TcPOU
// 隐含生成代码：不要编辑
FUNCTION CheckRangeSigned : DINT
VAR_INPUT
	value, lower, upper: DINT;
END_VAR

// 隐含生成代码：这里只是对代码实现的建议
{noflow}
IF (value < lower) THEN
	CheckRangeSigned := lower;
ELSIF(value > upper) THEN
	CheckRangeSigned := upper;
ELSE
	CheckRangeSigned := value;
END_IF
{flow}

END_FUNCTION

// ---- POUs/POUCheck/CheckRangeUnsigned.TcPOU
// 隐含生成代码：不要编辑
FUNCTION CheckRangeUnsigned : UDINT
VAR_INPUT
	value, lower, upper: UDINT;
END_VAR

// 隐含生成代码：这里只是对代码实现的建议
{noflow}
IF (value < lower) THEN
	CheckRangeUnsigned := lower;
ELSIF(value > upper) THEN
	CheckRangeUnsigned := upper;
ELSE
	CheckRangeUnsigned := value;
END_IF
{flow}

END_FUNCTION

// ---- GlobalTextList.TcGTLO
TEXTLIST GlobalTextList
  888 = '%d'
  896 = '%s'
  722 = 'Abort'
  14 = 'Aborted'
  193 = 'Aborting'
  503 = 'ABSPos: %f'
  412 = 'actPos: %f'
  242 = 'ActPos: %f'
  251 = 'ActTorq: %f'
  148 = 'ActTorque: %f'
  446 = 'ActTrquo: %f'
  498 = 'ActVel: %f'
  542 = 'ADDPos: %f'
  711 = 'AxisNo: %D'
  312 = 'AxisNo: %d'
  330 = 'CamIn'
  460 = 'CamOut'
  567 = 'Clear'
  38 = 'CLEAR        FAULT'
  225 = 'CLEAR FAULT'
  981 = 'ClearFault'
  670 = 'CLEARFAULT'
  75 = 'Clearing'
  183 = 'Cleat'
  579 = 'Complete'
  512 = 'completing'
  605 = 'Completing'
  679 = 'ENA'
  115 = 'ENABLE'
  359 = 'ERROR'
  425 = 'Execute'
  815 = 'Held'
  685 = 'Hold'
  625 = 'HOLD'
  465 = 'Holding'
  173 = 'HOME'
  142 = 'idel'
  48 = 'idle'
  669 = 'INGEAR'
  630 = 'INSYNC'
  761 = 'INVEL'
  563 = 'INVELO'
  918 = 'JOG'
  375 = 'Jog +'
  398 = 'Jog -'
  823 = 'Jog+'
  949 = 'Jog-'
  198 = 'JogN'
  24 = 'JogP'
  796 = 'JogVEL: %f'
  27 = 'MoveABS'
  245 = 'MoveAdd'
  522 = 'MoveADD'
  754 = 'MoveVEL'
  156 = 'MoveVel'
  756 = 'Pos: %f'
  494 = 'Reset'
  708 = 'RESET'
  96 = 'Resetting'
  799 = 'SafetyReset'
  504 = 'Start'
  773 = 'START'
  73 = 'Starting'
  733 = 'Stop'
  482 = 'STOP'
  743 = 'Stopped'
  324 = 'Stopping'
  361 = 'Suspend'
  334 = 'Suspended'
  107 = 'Suspending'
  942 = 'Unhold'
  843 = 'UnSuspe'
  4 = 'Unsuspend'
  935 = 'Uold'
  906 = 'VEL: %f'
  622 = '伺服编号: %d'
  95 = '使能'
  246 = '使能反馈'
  463 = '停止'
  760 = '凸轮同步'
  296 = '原点偏移: %f'
  769 = '原点反馈'
  295 = '反向点动'
  908 = '同步反馈'
  364 = '回零'
  730 = '复位'
  914 = '当前位置: %f'
  518 = '当前转速: %f'
  874 = '当前速度: %f'
  273 = '故障代码: %D'
  978 = '故障代码: %d'
  763 = '故障代码: %f'
  616 = '故障反馈'
  311 = '正向点动'
  167 = '点动速度: %f'
  923 = '目标位置: %f'
  445 = '相对定位'
  391 = '绝对定位'
  785 = '耦合反馈'
  794 = '解除凸轮'
  770 = '解除同步'
  757 = '解除同步轮'
  176 = '解除齿轮'
  253 = '速度模式'
  189 = '速度模式反馈'
  63 = '速度模式运行'
  527 = '速度设置: %f'
  131 = '速度运行'
  741 = '齿轮同步'
END_TEXTLIST

// ---- VISUs/EM.TcVIS
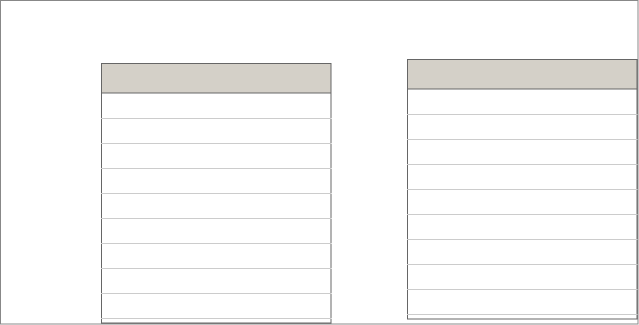
VISUALIZATION EM  // 639x325
    Table (101,63 230x260), data array: Unit01.EM_Resetting_Done
        p3854506369: Unit01.EM_Resetting_Done[INDEX]
    Table (407,59 230x260), data array: Unit02.EM_Resetting_Done
        p3854506369: Unit02.EM_Resetting_Done[INDEX]
END_VISUALIZATION

// ---- VISUs/Part/Visualization_Cnt.TcVIS
VISUALIZATION Visualization_Cnt  // 2x2
END_VISUALIZATION

// ---- VISUs/Part/Vis_Axis.TcVIS
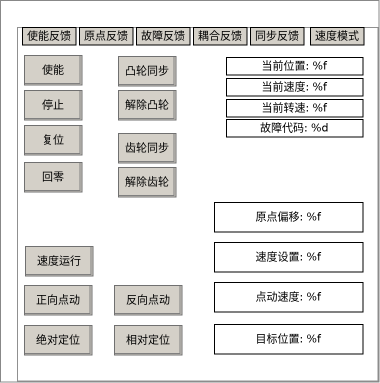
VISUALIZATION Vis_Axis  // 380x383
VAR_IN_OUT
	Axis:REFERENCE TO UDT_axisAdmin;
END_VAR
    GroupBox (17,19 361x362)
        Button (7,36 58x30), "使能"
            toggle Axis.i.Enable
        Button (8,227 68x30), "速度运行"
            tap Axis.i.MoveVel
        Button (101,37 58x30), "凸轮同步"
            tap Axis.i.CamIn
        Button (101,71 58x30), "解除凸轮"
            tap Axis.i.CamOut
        Button (7,71 58x30), "停止"
            tap Axis.i.Stop
        Button (7,106 58x30), "复位"
            tap Axis.i.Reset
        RoundedRectangle (209,38 137x18), "当前位置: %f", text variable: Axis.o.ActPos
        Button (7,266 68x30), "正向点动"
            tap Axis.i.JogP
        Button (97,266 68x30), "反向点动"
            tap Axis.i.JogN
        Rectangle (5,8 54x18), "使能反馈", colour toggle: Axis.o.PowerOn
        Rectangle (62,8 54x18), "原点反馈", colour toggle: Axis.o.Homed
        Rectangle (119,8 54x18), "故障反馈", colour toggle: Axis.o.Error
        Rectangle (176,8 54x18), "耦合反馈", colour toggle: Axis.o.InGear
        Rectangle (233,8 54x18), "同步反馈", colour toggle: Axis.o.InSync'
        Rectangle (293,8 54x18), "速度模式", colour toggle: Axis.o.InVelocity
        RoundedRectangle (209,59 137x18), "当前速度: %f", text variable: Axis.o.ActVel
        RoundedRectangle (209,80 137x18), "当前转速: %f", text variable: Axis.o.ActTorq
        Button (7,306 68x30), "绝对定位"
            tap Axis.i.MoveAbs
        Button (97,306 68x30), "相对定位"
            tap Axis.i.MoveAdd
        RoundedRectangle (197,263 149x30), "点动速度: %f", text variable: Axis.i.JogVel
            OnMouseClick: write the text variable via Default
        RoundedRectangle (197,305 149x30), "目标位置: %f", text variable: Axis.i.Pos
            OnMouseClick: write the text variable via Default
        RoundedRectangle (197,223 149x30), "速度设置: %f", text variable: Axis.i.Vel
            OnMouseClick: write the text variable via Default
        Button (101,148 58x30), "解除齿轮"
            tap Axis.i.GearOut
        RoundedRectangle (209,100 137x18), "故障代码: %d", text variable: Axis.o.ErrorID
        Button (7,143 58x30), "回零"
            tap Axis.i.Home
        RoundedRectangle (197,183 149x30), "原点偏移: %f", text variable: Axis.i.HomeOffset
            OnMouseClick: write the text variable via Default
    Button (118,133 58x30), "齿轮同步"
        tap Axis.i.GearIn
END_VISUALIZATION

// ---- VISUs/Part/Vis_PackMlv3.TcVIS
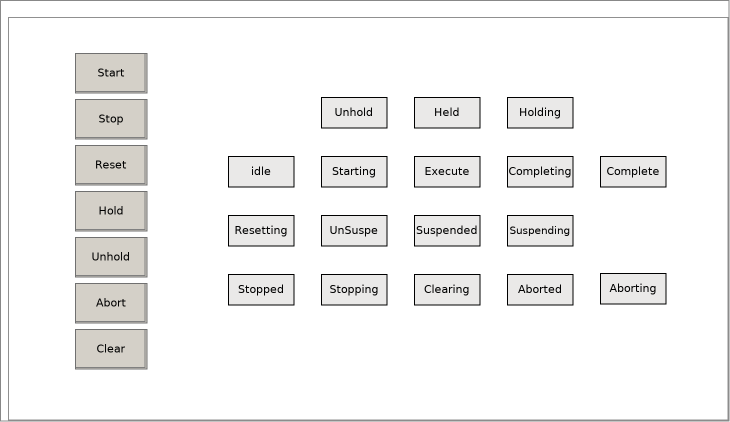
VISUALIZATION Vis_PackMlv3  // 730x422
VAR_IN_OUT
	PML3: PackMlv3_StateModel;
END_VAR
    GroupBox (8,9 720x411)
        RoundedRectangle (220,147 66x31), "idle", colour toggle: PML3.Sts_Idle
        Button (67,44 72x40), "Start"
            tap PML3.Cmd_Start
        Button (67,90 72x40), "Stop"
            tap PML3.Cmd_Stop
        Button (67,136 72x40), "Reset"
            tap PML3.Cmd_Reset
        Button (67,182 72x40), "Hold"
            tap PML3.Cmd_Hold
        Button (67,228 72x40), "Unhold"
            tap PML3.Cmd_UnHold
        Button (67,320 72x40), "Clear"
            tap PML3.Cmd_Clear
        Button (67,274 72x40), "Abort"
            tap PML3.Cmd_Abort
        RoundedRectangle (313,147 66x31), "Starting", colour toggle: PML3.Sts_Starting
        RoundedRectangle (406,147 66x31), "Execute", colour toggle: PML3.Sts_Execute
        RoundedRectangle (499,147 66x31), "Completing", colour toggle: PML3.Sts_Completing
        RoundedRectangle (592,147 66x31), "Complete", colour toggle: PML3.Sts_Complete
        RoundedRectangle (220,206 66x31), "Resetting", colour toggle: PML3.Sts_Resetting
        RoundedRectangle (313,88 66x31), "Unhold", colour toggle: PML3.Sts_UnHolding
        RoundedRectangle (220,265 66x31), "Stopped", colour toggle: PML3.Sts_Stopped
        RoundedRectangle (592,264 66x31), "Aborting", colour toggle: PML3.Sts_Aborting
    RoundedRectangle (321,215 66x31), "UnSuspe", colour toggle: PML3.Sts_UnSuspending
    RoundedRectangle (414,215 66x31), "Suspended", colour toggle: PML3.Sts_Suspended
    RoundedRectangle (507,215 66x31), "Suspending", colour toggle: PML3.Sts_Suspending
    RoundedRectangle (414,97 66x31), "Held", colour toggle: PML3.Sts_Held
    RoundedRectangle (507,97 66x31), "Holding", colour toggle: PML3.Sts_Holding
    RoundedRectangle (321,274 66x31), "Stopping", colour toggle: PML3.Sts_Stopping
    RoundedRectangle (414,274 66x31), "Clearing", colour toggle: PML3.Sts_Clearing
    RoundedRectangle (507,274 66x31), "Aborted", colour toggle: PML3.Sts_Aborted
END_VISUALIZATION

// ---- VISUs/Vis_MAIN.TcVIS
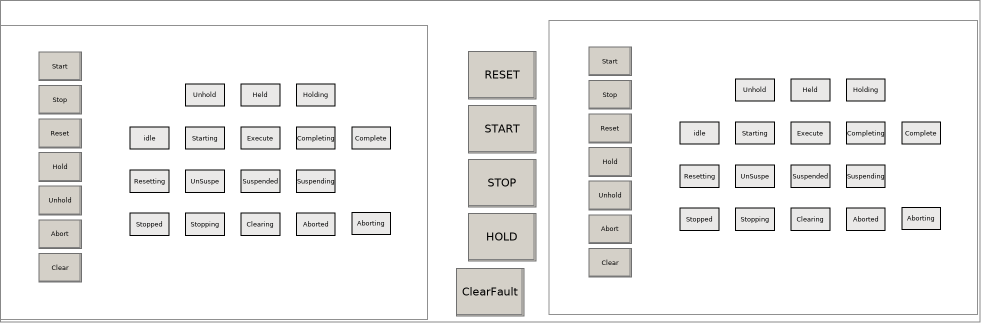
VISUALIZATION Vis_MAIN  // 981x323
    Frame (-6,13 435x308)
        shows Vis_PackMlv3(PML3 := UN01_MachineStateModel)
    Button (468,51 68x48), "RESET"
        tap HMI_Input.Reset
    Button (468,105 68x48), "START"
        tap HMI_Input.Start
    Button (468,159 68x48), "STOP"
        tap HMI_Input.Stop
    Button (468,213 68x48), "HOLD"
        tap HMI_Input.Hold
    Button (456,268 68x48), "ClearFault"
        tap UN01.xDebugReset
    Frame (544,8 435x308)
        shows Vis_PackMlv3(PML3 := UN02_MachineStateModel)
END_VISUALIZATION

// ---- VISUs/Vis_RealAxis.TcVIS
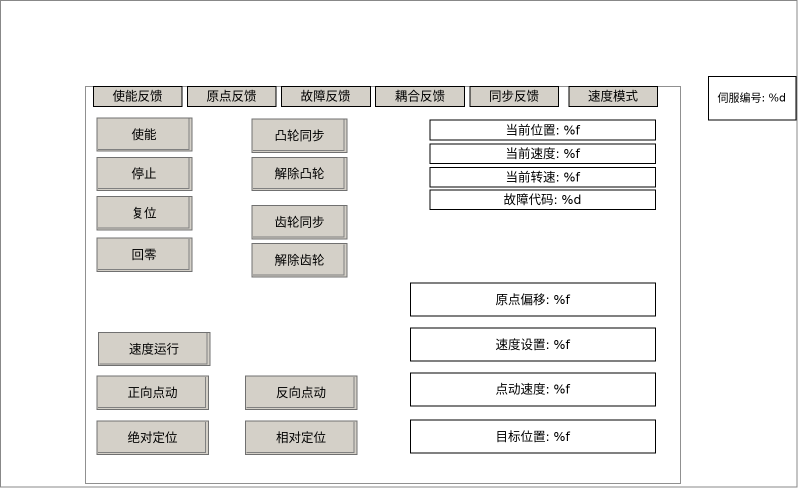
VISUALIZATION Vis_RealAxis  // 798x488
    Frame (57,56 627x430)
        shows Vis_Axis(Axis := MotionControl.Vis_RealAxisRef)
    Rectangle (708,76 88x44), "伺服编号: %d", text variable: MotionControl.Vis_RealAxisNoRef
        OnMouseClick: write the text variable via Default
END_VISUALIZATION

// ---- VISUs/Vis_VirtualAxis.TcVIS
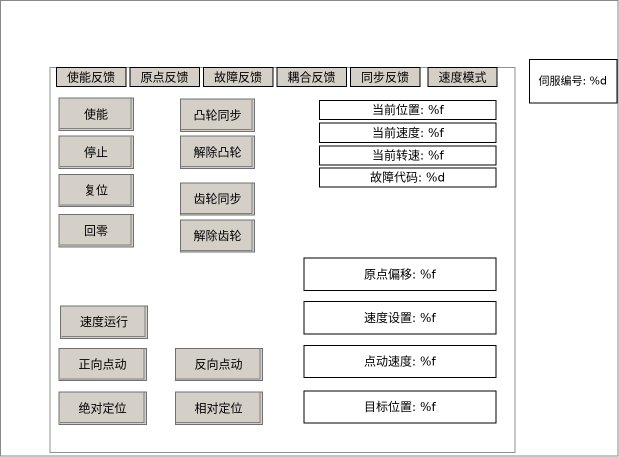
VISUALIZATION Vis_VirtualAxis  // 619x457
    Frame (28,38 490x417)
        shows Vis_Axis(Axis := MotionControl.Vis_VirtualAxisRef)
    Rectangle (529,59 88x44), "伺服编号: %d", text variable: MotionControl.Vis_VirtualAxisNoRef
        OnMouseClick: write the text variable via Default
END_VISUALIZATION
